// Inherit from this FB to get Tc2_System.ST_AmsAddr in the process image (to link to EtherCAT devices etc...)
FUNCTION_BLOCK ABSTRACT FB_HasAmsAddressFromProcessImage
VAR_INPUT
END_VAR
VAR_OUTPUT
END_VAR
VAR
	Ams AT%I* 	: Tc2_System.ST_AmsAddr;
	_ams 		: Tc2_System.ST_AmsAddr;
END_VAR

(* Gets or sets the Ams address structure*)
PROPERTY AmsAddress : REFERENCE TO Tc2_System.ST_AmsAddr
GET
_ams := Ams;
AmsAddress REF= _ams;
END_GET
END_PROPERTY

END_FUNCTION_BLOCK

(* stored: Version 1.1.0.1, ProductVersion 3.1.4024.14
   POU FB_HasAmsAddressFromProcessImage: Id {24569db7-6441-041f-19dc-eb8a43d6dd89}, SpecialFunc None
   Property AmsAddress: Id {87db1621-978a-01be-36e4-0f46484bdbe2}
   Get Get: Id {639bd165-9b0f-03a4-27a2-92e46b7d7dbb} *)
